FUNCTION_BLOCK RobotCustomPattern
VAR_INPUT
	ENI				: BOOL;
	CycleAtLayer	: UINT;
	dtRecipe		: stProductinfo;
END_VAR
VAR_OUTPUT
	ENO				: BOOL;
	Offset_X		: UINT;
	Offset_Y		: UINT;
	Offset_Z		: UINT;
END_VAR

VAR
	
END_VAR

IF ENI THEN
	ENO:=TRUE;
	
	
	IF CycleAtLayer <> 0 THEN
		Offset_X := INT_TO_UINT(dtRecipe.OffsetPattern.Offset_X[CycleAtLayer]);
		Offset_Y := INT_TO_UINT(dtRecipe.OffsetPattern.Offset_Y[CycleAtLayer]);
		Offset_Z := INT_TO_UINT(dtRecipe.OffsetPattern.Offset_Z[CycleAtLayer]);
	END_IF
	
	
	
END_IF;

END_FUNCTION_BLOCK

(* stored: Version 1.1.0.1, ProductVersion 3.1.4024.12
   POU RobotCustomPattern: Id {fcd1fbe7-c892-4392-9af5-2d5eec7f4aa5}, SpecialFunc None *)
